// TIA Portal V20 export
ORGANIZATION_BLOCK "Main"   // OB1, SCL, ProgramCycle
TITLE = "Main Program Sweep (Cycle)"
{ S7_Optimized_Access := 'TRUE' }
// stored: SetENOAutomatically false
   VAR_INPUT
      Initial_Call : Bool;   // Initial call of this OB
      Remanence : Bool;   // =True, if remanent data are available
   END_VAR
BEGIN
   REGION Description head
       //==================================================================================
       // POSALUX Swiss SA / (C) Copyright 2025
       //----------------------------------------------------------------------------------
       // Title: Main
       // Comment/Function: Cyclical execution of the program by the PLC
       // Author: Fabien WALDT
       // Engineering: TIA Portal v19
       //----------------------------------------------------------------------------------
       // Change log table:
       // Version  | Date     | Expert in charge | Changes applied
       //----------------------------------------------------------------------------------
       // 00.00.01 | 20250423 | WFA              | First released version
       //==================================================================================
   END_REGION

   REGION CNC
       // Call block for cyclical data exchange NC <-> PLC for the MCP
       "LBP_OpUnitComm_DB"(Config := "LBP_ConfigData");
       "LBP_MainBP"();
   END_REGION

   REGION IO
       "FC_AnalogInputsInit"();
       "DB_AnalogInputs"();
       "FC_AnalogInputAction"(iReset := "DB_McpKeyboardSignals".sAlarmReset.sKeySWStatus OR "MCP1_In".reset,
                              oBadPartOnFixture => "DB_BadPartOnFixture".BadPartOnFixture,
                              oID_MeasureBad=>"DB_BadPartOnFixture".ID_MeasureBad);
       "FC_AnalogInputConfig"();
       "DB_DigitalInputs"();
       "DB_DigitalInputsSonplas"();
       "DB_DigitalInputsBW_Station"();

       "DB_AnalogOutputs"();
       "DB_DigitalOutputs"();
       "DB_DigitalOutputsSonplas"();  
   END_REGION

   REGION Basic fonctions
       "DB_Impulsion"();
       "DB_ReadDateAndTime"();
   END_REGION

   REGION Interface PLC_ISO
       "DB_CommPLC_ISO"();
       "DB_MiscPLC_IHM_ISO"();
   END_REGION

   REGION SAFETY
       "FC_DataToSafety"();
       "DB_Alarms_Safety"();
   END_REGION

   REGION Load Unload Parts
       "DB_LoaderMain"();
       "DB_LoaderFixtureMain"();
       "DB_ExtraMissingPart"();
       "DB_PrioSequence"();
   END_REGION

   REGION Alarms
       "DB_Alarms"();

       "LBP_GenerateAlarmMsgs"(ToUserIF := true,
                               Quit := true,
                               NumActAlarmMsgs => "LBP_ConfigData".GenerateAlarmMsgs.NumActAlarmMsgs,
                               Error => "LBP_ConfigData".GenerateAlarmMsgs.Error,
                               StatusID => "LBP_ConfigData".GenerateAlarmMsgs.StatusID,
                               Status => "LBP_ConfigData".GenerateAlarmMsgs.Status);
       "DB_Msg"();
   END_REGION

   REGION Base Machine
       REGION Channel
           "DB_DecodChannels"();
           "DB_CycleStartStop"();
        END_REGION   

        REGION Axis
            "DB_Axis"();
            "DB_AxisPosition"();
        END_REGION

        REGION MCP
            "DB_MCPManagement"(); // Must be called after FC10 (LBP_GenerateAlarmMsgs)
        END_REGION

        REGION Laser
            "DB_LaserAirProcess"();
            "DB_LaserOperation"();
            "DB_LaserMeasureZoneSwitch"();  // WFA A Confirmer si plus utilisé
            "DB_Powermeter"();
        END_REGION

        REGION Air system
            "DB_Pressures"();
            "DB_Vacuums"();
        END_REGION

       REGION Vision
           "DB_Cognex"();
       END_REGION

       REGION Power Management
           "DB_Machineshutdown_UPS"();
           "DB_PowerOn"();
       END_REGION

       REGION Maintenance
           "DB_Maintenances"();
       END_REGION

       REGION Temperature Management
           "DB_Temperature"();
           "FC_ChillerMain"();
       END_REGION

       REGION Warm Up
           "DB_WarmUP"();
       END_REGION

       REGION Feed Override Display
           "DB_FeedOverride"(iA_FD_OR:="LBP_Chan1".A_FD_OR,
                             oFeedOverride=>"DB_FeedOverride".oFeedOverride);

       END_REGION
   END_REGION

   REGION Lights Management
       "DB_LightsManagement"();
   END_REGION

   REGION Main Door Management
       "DB_MainDoorManagement"();
   END_REGION

   REGION Config Machine
       "FC_GestionConfigMachine"();
   END_REGION

   REGION Tracability
       "DB_Tracability"(iCondTransfertExtInTo1:="DB_PartManagement".sPosition.sShuttle1.Undrilled.Presence.Part,
                        iCondTransfertExtInTo2:="DB_PartManagement".sPosition.sShuttle2.Undrilled.Presence.Part,
                        iCondTransfert1To3:="DB_LoaderShuttle1".sIntLoadUnload.oLoadGripperCloseReq,
                        iCondTransfert2To3:="DB_LoaderShuttle2".sIntLoadUnload.oLoadGripperCloseReq,
                        iCondTransfert3To4:="DB_PartManagement".sPosition.sFixture.Undrilled.Presence.Part,
                        iCondTransfert4To5:="DB_PartManagement".sPosition.sGripper.Drilled.Presence.Part,
                        iCondTransfert5To6:="DB_LoaderShuttle1".sIntLoadUnload.oUnloadGripperOpenReq,
                        iCondTransfert5To7:="DB_LoaderShuttle2".sIntLoadUnload.oUnloadGripperOpenReq,
                        iCondTransfert6ToExtOut:="DB_LoaderShuttle1".sExtLoadUnload.sInterface.JobDone AND NOT "DB_WorkingModes".sFilling,
                        iCondTransfert7ToExtOut:="DB_LoaderShuttle2".sExtLoadUnload.sInterface.JobDone AND NOT "DB_WorkingModes".sFilling);
   END_REGION

   REGION External Loader
       "DB_SonplasMain"();
   END_REGION

   REGION OPC
       // Keys
       "DB_HmiKeyboardSignals"();

       // Machine
       "DB_Parameters"();

       // Axis
       "DB_OPC_AxisManagement"();

       // State
       "DB_OPC_State"();

       // RealTime
       "DB_RealTime"();

       // Components
       "DB_Components"();

       // Laser
       "DB_Scanner"();
       "DB_Part_Data"();

       // Recipe
       "DB_Recipe"();
   END_REGION

   REGION Part Management
       "DB_PartManagement"();
   END_REGION

   REGION Bw loader
       "DB_BwLoader"();

   END_REGION

   REGION Working Modes
       "DB_GestionWorkingModes"();
   END_REGION

   REGION WAF A SUPPRIMER
       "DB_Simulation"();
   "DB_HMI_PLC_Pos"("HMI_Change Enable":=FALSE,
                    ioPLC_State:="DB_WAF".PLC_Pos,
                    ioHMI_State:="DB_WAF".HMI_Pos);
   END_REGION
END_ORGANIZATION_BLOCK
